# EPICS substitutions: db/Beckhoff_2XXX/ecmcEPP2008.substitutions
# generic slave part
file "ecmcEcSlave.template"{
  pattern {}
          {}
}

# binary outputs
file "ecmc_binaryOutput-chX.template"{
  pattern {CH_ID}
          {01   }
          {02   }
          {03   }
          {04   }
          {05   }
          {06   }
          {07   }
          {08   }
}
